PROGRAM MAIN
VAR
VesselControll_Program :	VesselControlFB ;
END_VAR

VesselControll_Program();

END_PROGRAM

(* stored: Version 1.1.0.1, ProductVersion 3.1.4024.12
   POU MAIN: Id {dc601566-8139-4f5a-b1ac-259dda6c5dad}, SpecialFunc None *)
